(* IEC 61131-3 sources: AutomationLab/ConveyerObject/Support, 5 files *)

(* ---- Conveyer_Hardware_FB.st ---- *)
FUNCTION_BLOCK Conveyer_Hardware_FB
VAR_INPUT
END_VAR
VAR_OUTPUT
END_VAR
VAR_IN_OUT
    Data: ConveyerType;
END_VAR

// Датчик оптический, нормально замкнутый:
// нет коробки — цепь замкнута (TRUE), коробка обнаружена — цепь разомкнута (FALSE)
// Инвертируем для получения логического состояния "коробка на конце"
Data.BoxOnEndPosition := NOT GVL.DI_SensorA;

// Запись команды двигателя в глобальную переменную
GVL.DO_ComMotor := Data.ComRotateLent;

(* ---- Conveyer_HardwareIn_FB.st ---- *)
FUNCTION_BLOCK Conveyer_HardwareIn_FB
VAR_INPUT
END_VAR
VAR_OUTPUT
END_VAR
VAR_IN_OUT
    Data: DT_Conveyer;
END_VAR
VAR
    sensorDebounce: TON;
END_VAR

// ВХОД: чтение оптического датчика (нормально замкнутого) с антидребезгом.
// Нет коробки — цепь замкнута (TRUE), коробка обнаружена — цепь разомкнута (FALSE).
// Инвертируем для получения логического состояния "коробка на конце".
sensorDebounce(IN := NOT GVL.DI_SensorA, PT := T#50ms);
Data.BoxOnEndPosition := sensorDebounce.Q;

(* ---- Conveyer_HardwareOut_FB.st ---- *)
FUNCTION_BLOCK Conveyer_HardwareOut_FB
VAR_INPUT
END_VAR
VAR_OUTPUT
END_VAR
VAR_IN_OUT
    Data: DT_Conveyer;
END_VAR

// ВЫХОД: запись команды двигателя в глобальную переменную
GVL.DO_ComMotor := Data.ComRotateLent;

(* ---- Conveyer_HMI_FB.st ---- *)
FUNCTION_BLOCK Conveyer_HMI_FB
VAR_INPUT
END_VAR
VAR_OUTPUT
END_VAR
VAR_IN_OUT
    Data: DT_Conveyer;
END_VAR

// Сигнализация работы конвейера — лампа для оператора
GVL.DO_LampWork := Data.ComRotateLent;

(* ---- Hardware.st ---- *)
FUNCTION_BLOCK Hardware
VAR_INPUT
	SensorA: BOOL;
END_VAR
VAR_OUTPUT
	ComMotor: BOOL;
END_VAR
VAR_IN_OUT
    Data: ConveyerType;
END_VAR

// Датчик оптический, нормально замкнутый:
// нет коробки — цепь замкнута (TRUE), коробка обнаружена — цепь разомкнута (FALSE)
// Инвертируем для получения логического состояния "коробка на конце"
Data.BoxOnEndPosition := NOT SensorA;

// Запись команды двигателя
ComMotor := Data.ComRotateLent;
